SUBAPPLICATION Wasserventil (* Steuert den digitalen Ausgang (MI_00 / DigitalOutput_5A) fuer das Wasserventil und meldet dessen Ist-Zustand sowie Status zurueck *)
  (* Standard: 61499-2 *)
  (* Version 1.0, 2024-04-23, Elias *)
  IMPORT DataPanel::io::MI::DQ::DataPanel_MI_DO::DigitalOutput_5A;
  IMPORT DataPanel::io::MI::const::MI::MI_00;
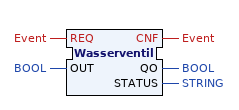
  EVENT_INPUT
    REQ; (* Anforderung: Ausgang gemaess OUT ansteuern *)
  END_EVENT
  EVENT_OUTPUT
    CNF; (* Bestaetigung: Ansteuerung abgeschlossen *)
  END_EVENT
  VAR_INPUT
    OUT : BOOL; (* Sollwert des Ausgangs (TRUE = Wasserventil geoeffnet) *)
  END_VAR
  VAR_OUTPUT
    QO : BOOL; (* Rueckgelesener Ist-Zustand des digitalen Ausgangs *)
    STATUS : STRING; (* Status-/Diagnosemeldung des digitalen Ausgangs *)
  END_VAR
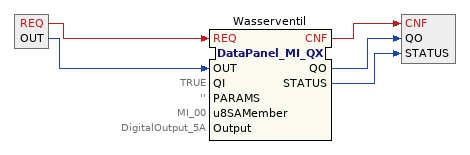
  FBS
    Wasserventil : DataPanel::io::MI::DQ::DataPanel_MI_QX(QI := TRUE, PARAMS := '', u8SAMember := MI_00, Output := DigitalOutput_5A);
  END_FBS
  EVENT_CONNECTIONS
    REQ TO Wasserventil.REQ;
    Wasserventil.CNF TO CNF;
  END_CONNECTIONS
  DATA_CONNECTIONS
    OUT TO Wasserventil.OUT;
    Wasserventil.QO TO QO;
    Wasserventil.STATUS TO STATUS;
  END_CONNECTIONS
END_SUBAPPLICATION
